(* PLC project Unnamed, Unknown Unnamed 1 *)
(* stored: creationDateTime 2013-01-29T14:01:00, modificationDateTime 2013-02-26T15:59:13 *)

TYPE LOGLEVEL : (CRITICAL, WARNING, INFO, DEBUG) := INFO;
END_TYPE

FUNCTION_BLOCK LOGGER
  VAR_INPUT
    TRIG : BOOL;
    MSG : STRING;
    LEVEL : LOGLEVEL := INFO;
  END_VAR
  VAR
    TRIG0 : BOOL;
  END_VAR

IF TRIG AND NOT TRIG0 THEN
{{
 LogMessage(GetFbVar(LEVEL),(char*)GetFbVar(MSG, .body),GetFbVar(MSG, .len));
}}
END_IF;
TRIG0:=TRIG;

          
END_FUNCTION_BLOCK

FUNCTION_BLOCK DISPLAYMESSAGES
  VAR_INPUT
    TRIG : BOOL;
    MSG1 : STRING;
    MSG2 : STRING;
    MSG3 : STRING;
  END_VAR
  VAR
    TRIG0 : BOOL;
    MSG : STRING;
  END_VAR

IF TRIG AND NOT TRIG0 THEN
MSG := CONCAT(MSG1, MSG2, MSG3);
{{
// DisplayMessages((char*)GetFbVar(MSG, .body), GetFbVar(MSG, .len), (char*)GetFbVar(MSG1, .body), GetFbVar(MSG1, .len), (char*)GetFbVar(MSG2, .body), GetFbVar(MSG2, .len));
  LogMessage(1, (char*)GetFbVar(MSG, .body), GetFbVar(MSG, .len));
}}
END_IF;
TRIG0:=TRIG;

          
END_FUNCTION_BLOCK

FUNCTION_BLOCK DISPLAYBUTTONS
  VAR_INPUT
    TRIG : BOOL;
    BTNTEXT1 : STRING;
    BTNCODE1 : INT;
    BTNTEXT2 : STRING;
    BTNCODE2 : INT;
    BTNTEXT3 : STRING;
    BTNCODE3 : INT;
  END_VAR
  VAR
    TRIG0 : BOOL;
    MSG : STRING;
    CODESTR1 : STRING;
    CODESTR2 : STRING;
    CODESTR3 : STRING;
  END_VAR

IF TRIG AND NOT TRIG0 THEN
CODESTR1 := INT_TO_STRING(BTNCODE1);
CODESTR2 := INT_TO_STRING(BTNCODE2);
CODESTR3 := INT_TO_STRING(BTNCODE3);
MSG := CONCAT('BUTTON1: ', BTNTEXT1, 'CODE1: ', CODESTR1, 'BUTTON2: ', BTNTEXT2, 'CODE2: ', CODESTR2, 'BUTTON3: ', BTNTEXT3, 'CODE3: ', CODESTR3);
{{
// DisplayButtons((char*)GetFbVar(BTNTEXT1, .body), GetFbVar(BTNTEXT1, .len), GetFbVar(BTNCODE1), (char*)GetFbVar(BTNTEXT2, .body), GetFbVar(BTNTEXT2, .len), GetFbVar(BTNCODE2), (char*)GetFbVar(BTNTEXT3, .body), GetFbVar(BTNTEXT3, .len), GetFbVar(BTNCODE3));
  LogMessage(1, (char*)GetFbVar(MSG, .body), GetFbVar(MSG, .len));
}}
END_IF;
TRIG0:=TRIG;

          
END_FUNCTION_BLOCK

FUNCTION_BLOCK BUTTONPRESSED
  VAR_INPUT
    TRIG : BOOL;
    PROCESSED : BOOL;
  END_VAR
  VAR_OUTPUT
    CODE : INT;
  END_VAR
  VAR
    TRIG0 : BOOL;
    MSG : STRING;
  END_VAR

IF TRIG AND NOT TRIG0 THEN
MSG := 'BUTTONPRESSED is processed.';
{{
//  ButtonProcessed(GetFbVar(PROCESSED));
  LogMessage(1, (char*)GetFbVar(MSG, .body), GetFbVar(MSG, .len));
}}
CODE := 0;
END_IF;
TRIG0:=TRIG;

          
END_FUNCTION_BLOCK
